// TIA Portal V16 export
// export: Created 2023-01-04T15:44:08.8830907Z, ExportSetting WithDefaults, DisplayName Totally Integrated Automation Portal, DisplayVersion V16, DisplayName TIA Portal Version Control Interface, DisplayVersion V16, DisplayName TIA Portal Openness, DisplayVersion V16, DisplayName STEP 7 Professional, DisplayVersion V16, DisplayName STEP 7 Safety, DisplayVersion V16, DisplayName WinCC Advanced, DisplayVersion V16
FUNCTION_BLOCK "Tank1"   // FB4, LAD
{ S7_Optimized_Access := 'TRUE' }
VERSION : 0.1
// stored: AutoNumber true, IsIECCheckEnabled false, IsRetainMemResEnabled false, MemoryReserve 100, SetENOAutomatically false, UDAEnableTagReadback false
   VAR_INPUT
      EN_1 : Bool;
   END_VAR
   VAR_TEMP   // added for the SCL form of the ladder/FBD networks
      _w1 : Bool;
      _w2 : Bool;
      _w3 : Bool;
   END_VAR
BEGIN

REGION Network 1: Filling Process from Tank1
   // 0-27648 to 0-250ml
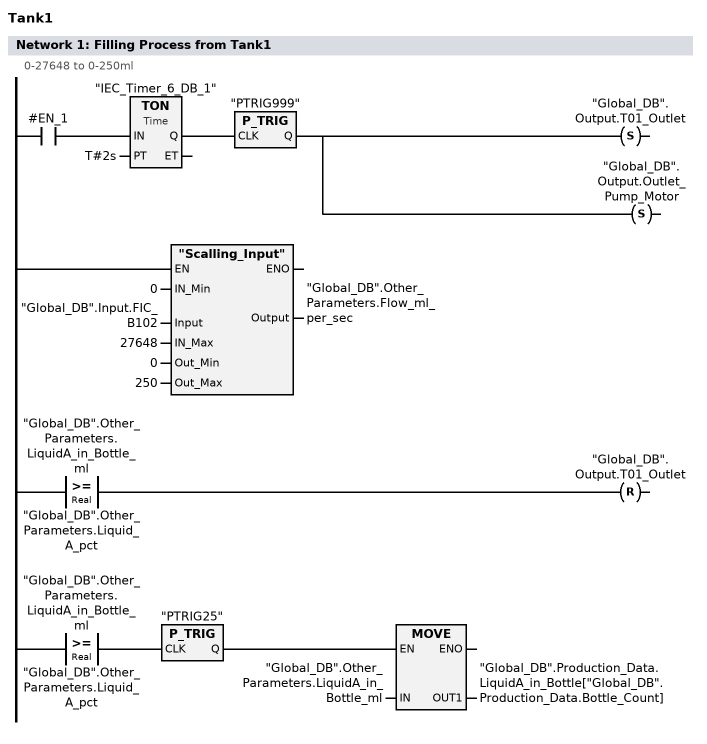
   RUNG wire#powerrail
      Contact( #EN_1 )
      { S7_Templates := "time_type := Time" } "IEC_Timer_6_DB_1".TON(pt := T#2s, et =>)
      P_Trig( "PTRIG999" )
      wire#w1
      S_Coil( "Global_DB".Output.T01_Outlet )
   END_RUNG
   RUNG wire#w1
      S_Coil( "Global_DB".Output.Outlet_Pump_Motor )
   END_RUNG
   RUNG wire#powerrail
      "Scalling_Input"(IN_Min := 0, Input := "Global_DB".Input.FIC_B102, IN_Max := 27648, Out_Min := 0, Out_Max := 250, Output => "Global_DB".Other_Parameters.Flow_ml_per_sec)
   END_RUNG
   RUNG wire#powerrail
      { S7_Templates := "SrcType := Real" } GE_Contact(in1 := "Global_DB".Other_Parameters.LiquidA_in_Bottle_ml, in2 := "Global_DB".Other_Parameters.Liquid_A_pct)
      R_Coil( "Global_DB".Output.T01_Outlet )
   END_RUNG
   RUNG wire#powerrail
      { S7_Templates := "SrcType := Real" } GE_Contact(in1 := "Global_DB".Other_Parameters.LiquidA_in_Bottle_ml, in2 := "Global_DB".Other_Parameters.Liquid_A_pct)
      P_Trig( "PTRIG25" )
      Move(in := "Global_DB".Other_Parameters.LiquidA_in_Bottle_ml, out1 => "Global_DB".Production_Data.LiquidA_in_Bottle["Global_DB".Production_Data.Bottle_Count])
   END_RUNG
   // the same network as SCL:
   "IEC_Timer_6_DB_1".TON(IN := #EN_1, PT := T#2s);
   #_w1 := "IEC_Timer_6_DB_1".Q AND NOT "PTRIG999";   // rising edge
   "PTRIG999" := "IEC_Timer_6_DB_1".Q;
   IF #_w1 THEN
       "Global_DB".Output.T01_Outlet := TRUE;
       "Global_DB".Output.Outlet_Pump_Motor := TRUE;
   END_IF;
   "Scalling_Input"(IN_Min := 0,
                    Input := "Global_DB".Input.FIC_B102,
                    IN_Max := 27648,
                    Out_Min := 0,
                    Out_Max := 250,
                    Output => "Global_DB".Other_Parameters.Flow_ml_per_sec);
   IF "Global_DB".Other_Parameters.LiquidA_in_Bottle_ml >= "Global_DB".Other_Parameters.Liquid_A_pct THEN
       "Global_DB".Output.T01_Outlet := FALSE;
   END_IF;
   #_w2 := "Global_DB".Other_Parameters.LiquidA_in_Bottle_ml >= "Global_DB".Other_Parameters.Liquid_A_pct;
   #_w3 := #_w2 AND NOT "PTRIG25";   // rising edge
   "PTRIG25" := #_w2;
   IF #_w3 THEN
       "Global_DB".Production_Data.LiquidA_in_Bottle["Global_DB".Production_Data.Bottle_Count] := "Global_DB".Other_Parameters.LiquidA_in_Bottle_ml;
   END_IF;
END_REGION
END_FUNCTION_BLOCK
